% RSLogix 500 project SARAN_TI_BAK036.RSS, saved by version 8.10.00.18 %
PROJECT "SARAN_TI"    % processor: MicroLogix 1200 %

PROGRAM FILES
  LAD 2   11 rungs

DATA FILES
  O0 OUTPUT  4 elements
  I1 INPUT  4 elements
  S2 STATUS  66 elements
  B3 BINARY  1 elements
  T4 TIMER  1 elements
  C5 COUNTER  3 elements
  R6 CONTROL  1 elements
  N7 INTEGER  1 elements

LADDER 2
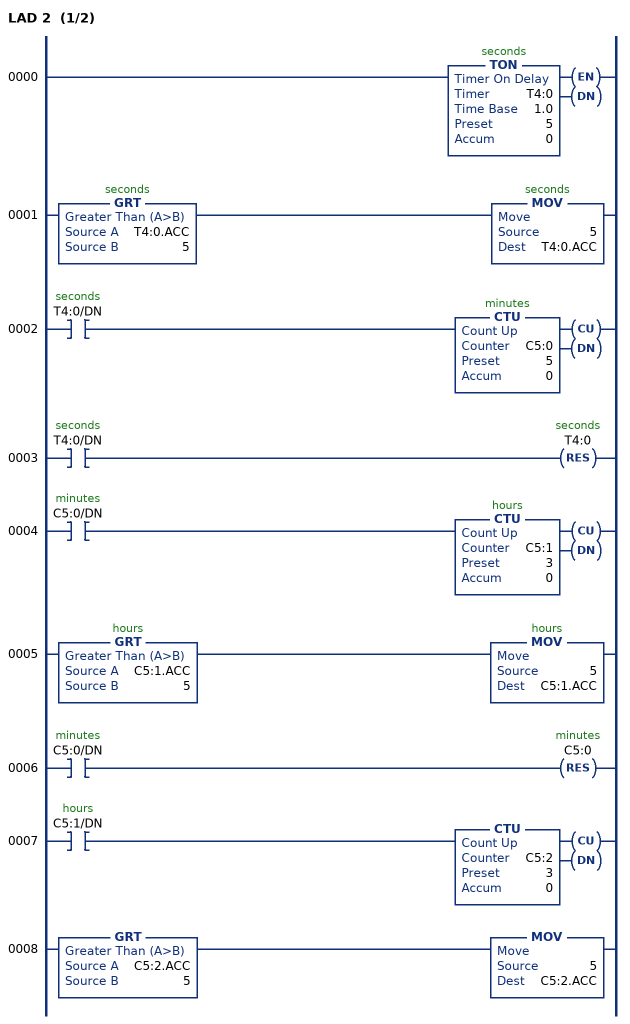
% Rung: 0 %
SOR TON T4:0 1.0 5 0 EOR
%   T4:0  "seconds" %
% Rung: 1 %
SOR GRT T4:0.ACC 5 MOV 5 T4:0.ACC EOR
%   T4:0  "seconds" %
% Rung: 2 %
SOR XIC T4:0/DN CTU C5:0 5 0 EOR
%   T4:0  "seconds" %
%   C5:0  "minutes" %
% Rung: 3 %
SOR XIC T4:0/DN RES T4:0 EOR
%   T4:0  "seconds" %
% Rung: 4 %
SOR XIC C5:0/DN CTU C5:1 3 0 EOR
%   C5:0  "minutes" %
%   C5:1  "hours" %
% Rung: 5 %
SOR GRT C5:1.ACC 5 MOV 5 C5:1.ACC EOR
%   C5:1  "hours" %
% Rung: 6 %
SOR XIC C5:0/DN RES C5:0 EOR
%   C5:0  "minutes" %
% Rung: 7 %
SOR XIC C5:1/DN CTU C5:2 3 0 EOR
%   C5:1  "hours" %
% Rung: 8 %
SOR GRT C5:2.ACC 5 MOV 5 C5:2.ACC EOR

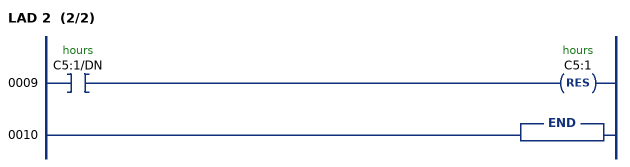
% Rung: 9 %
SOR XIC C5:1/DN RES C5:1 EOR
%   C5:1  "hours" %
% Rung: 10 %
SOR END EOR

DATA TABLE (non-zero values as saved)
DATA T4
% .PRE .ACC %
% T4:0 % 5 0
DATA C5
% .PRE .ACC %
% C5:0 % 5 0
% C5:1 % 3 0
% C5:2 % 3 0
